Staubli VAL3: placePlate.pgx

public program placePlate(num nPlate (dimensions=1))
begin
  //ADJUSTMENT: chance goHotel argument
  //when test phase is over (0 to 1)
  //robot supposed to be at Beam (goHotel(1))
  call goHotel(1)
  movel(appro(pHotel[nHoldingPlate],trPickPlateHor),flange,mNomSpeed)
  movel(appro(pHotel[nHoldingPlate],trPickPlateVer),flange,mNomSpeed)
  movel(pHotel[nHoldingPlate],flange,mNomSpeed)
  open(flange)
  delay(1)
  movel(appro(pHotel[nHoldingPlate],trPickPlateVer),flange,mNomSpeed)
  movel(appro(pHotel[nHoldingPlate],trPickPlateHor),flange,mNomSpeed)
  movel(pHotel[0],flange,mNomSpeed)
  waitEndMove()
  nHoldingPlate=0
end
